FUNCTION derivcvar_c: REAL
{ S7_Optimized_Access := 'false' }
    VAR_INPUT
        state: STATE;
    END_VAR

BEGIN
    derivcvar_c := state.cvar_c;
END_FUNCTION
